PROGRAM ArrayStorage
VAR
	aPotValues : ARRAY [lowBound..highBound] OF INT ;
	i: INT :=1;
	ftrig1: F_TRIG;
	rtrig1: R_TRIG;
END_VAR

VAR CONSTANT
	lowBound : 	INT := 1;
	highBound : INT := 5;
END_VAR

IF GVL.aSwitches[1] AND i>=lowBound AND i<=highBound THEN 
	aPotValues[i] := GVL.iPot1;
END_IF

ftrig1(CLK:= GVL.aSwitches[1]);


IF ftrig1.Q AND i>=lowBound AND i<highBound THEN
	i := i+1;
END_IF

IF gvl.bReset THEN
	FOR i:= lowBound TO highBound DO
		aPotValues[i] := 0;
	END_FOR
	i := lowBound;
	END_IF
	
rtrig1(CLK:= GVL.aSwitches[2]);
	
IF rtrig1.Q THEN
	i := i-1;
	IF i>= lowBound AND i<= highBound THEN
		aPotValues[i] := 0;
	END_IF
	IF i < lowBound THEN
		i := lowBound;
	END_IF
END_IF

END_PROGRAM

(* stored: Version 1.1.0.1, ProductVersion 3.1.4024.12
   POU ArrayStorage: Id {214e300a-074e-4623-b554-222b752a279c}, SpecialFunc None *)
